TYPE ST_VRC_NO EXTENDS ST_ValveBase:
STRUCT
(* Readbacks *)
	//In case VRC is normally open
	{attribute 'pytmc' := '
    pv: CLS_OK;
	field: ONAM CLOSE; 
	field: ZNAM OPEN;
	io: i;
    '}
	xCLS_OK : BOOL := TRUE;
	{attribute 'pytmc' := '
	pv: CLS_SW ;
	field: ONAM CLOSE; 
	field: ZNAM OPEN;
	io: io ;
	'}
	pv_xCLS_SW	: BOOL;
	{attribute 'pytmc' := '
    pv: FORCE_CLS;
	field: ONAM CLOSE; 
	field: ZNAM OPEN;
	io: io;
	'}
	pv_xOvrdCls	:	BOOL;

END_STRUCT
END_TYPE

(* stored: Version 1.1.0.1, ProductVersion 3.1.4022.18
   DUT ST_VRC_NO: Id {c04e91ec-1330-4fa3-ab98-dde61979a06a} *)
